PROGRAM OP20_Initialization_Seq
VAR
END_VAR

IF (SR20_Vert_servo_ctrl.Axis_In_Home)THEN
OP20_Temp_hmeOK:=TRUE;
OP20_HomeRunning:=FALSE;
OP20_Homing_Seq:=0;
ELSE
	OP20_Temp_hmeOK:=FALSE;	
END_IF

CASE OP20_Homing_Seq OF
	0: IF (OP20_AutoSelected AND NOT OP20_HomeRunning AND NOT OP20_ErrorActive AND NOT OP20_AutoRunning AND NOT OP20_StepRunning AND NOT OP20_Temp_hmeOK) THEN
		OP20_HomeRunning:=TRUE;
		OP20_Homing_Seq:=10;	
	   END_IF
	10:IF (OP20_HomeRunning AND (OP20_HMI_Homing OR HMI_Reset))THEN 
			IF (SR20_Vert_servo_ctrl.Axis_In_Home) THEN 
				//OP20_Homing_Seq:=20;
				SR20_Vert_servo_ctrl.Axis_Home_Cmd:=FALSE;
			ELSE
				SR20_Vert_servo_ctrl.Position:=0;
				SR20_Vert_servo_ctrl.Velocity:=100;
				SR20_Vert_servo_ctrl.ABSmove_Start:=TRUE;
				SR20_Vert_servo_ctrl.Axis_Home_Cmd:=TRUE;
	    	END_IF
			IF SR20_Vert_servo_ctrl.Axis_In_Home THEN
			  OP20_Homing_Seq:=20;			
			END_IF
	   END_IF		
	20:	OP20_Homing_Seq:=0;
		OP20_HomeRunning:=FALSE;
		OP20_HMI_Homing:=FALSE;
END_CASE

END_PROGRAM

(* stored: Version 1.1.0.1, ProductVersion 3.1.4024.11
   POU OP20_Initialization_Seq: Id {1637b520-7386-4833-96db-078875051f70}, SpecialFunc None *)
